
// ===== library: MasterCopy "maniobra_secado" =====

FUNCTION_BLOCK "maniobra_secado"   // FB3, STL
{ S7_Optimized_Access := 'TRUE' }
VERSION : 0.1
BEGIN
END_FUNCTION_BLOCK

// ===== library: MasterCopy "maniobra_pickandplace" =====

FUNCTION_BLOCK "maniobra_pickandplace"   // FB4, STL
{ S7_Optimized_Access := 'TRUE' }
VERSION : 0.1
BEGIN
END_FUNCTION_BLOCK